FUNCTION_BLOCK FB_NTZ_KW
VAR_INPUT
	Freigabe_auto			: BOOL;
	Freigabe_Deakt_auto		: BOOL;
	Betrieb_Anford_auto		: BOOL;
	Regelung_Modus_auto		: SINT;
	Regelung_Sollw_auto		: REAL;
	Zustand_PSp				: ST_PSp_Zustand;
END_VAR
VAR_OUTPUT
END_VAR
VAR
	{attribute 'OPC.UA.DA' := '1'}Steuerung				: ST_ThNTZ_Steuerung;		
	{attribute 'OPC.UA.DA' := '1'}Stellwert				: ST_ThNTZ_Stellwert;		
	{attribute 'OPC.UA.DA' := '1'}Zustand					: ST_ThNTZ_Zustand;		
	{attribute 'OPC.UA.DA' := '1'}Parameter				: ST_ThNTZ_Parameter;		

	Zuweisungen             : FB_KW_Zuweisungen;
	Zustandscheck			: FB_ThNTZ_Zustandscheck;
	Logik					: FB_ThNTZ_Logik;
	Ablaufsteuerung			: FB_ThNTZ_Ablaufsteuerung;
	Sollwertscheck			: FB_ThNTZ_Sollwertscheck;
	Regelung				: FB_ThNTZ_Regelung_Kaltnetz;
	Stellwertscheck			: FB_ThNTZ_Stellwertscheck;
END_VAR

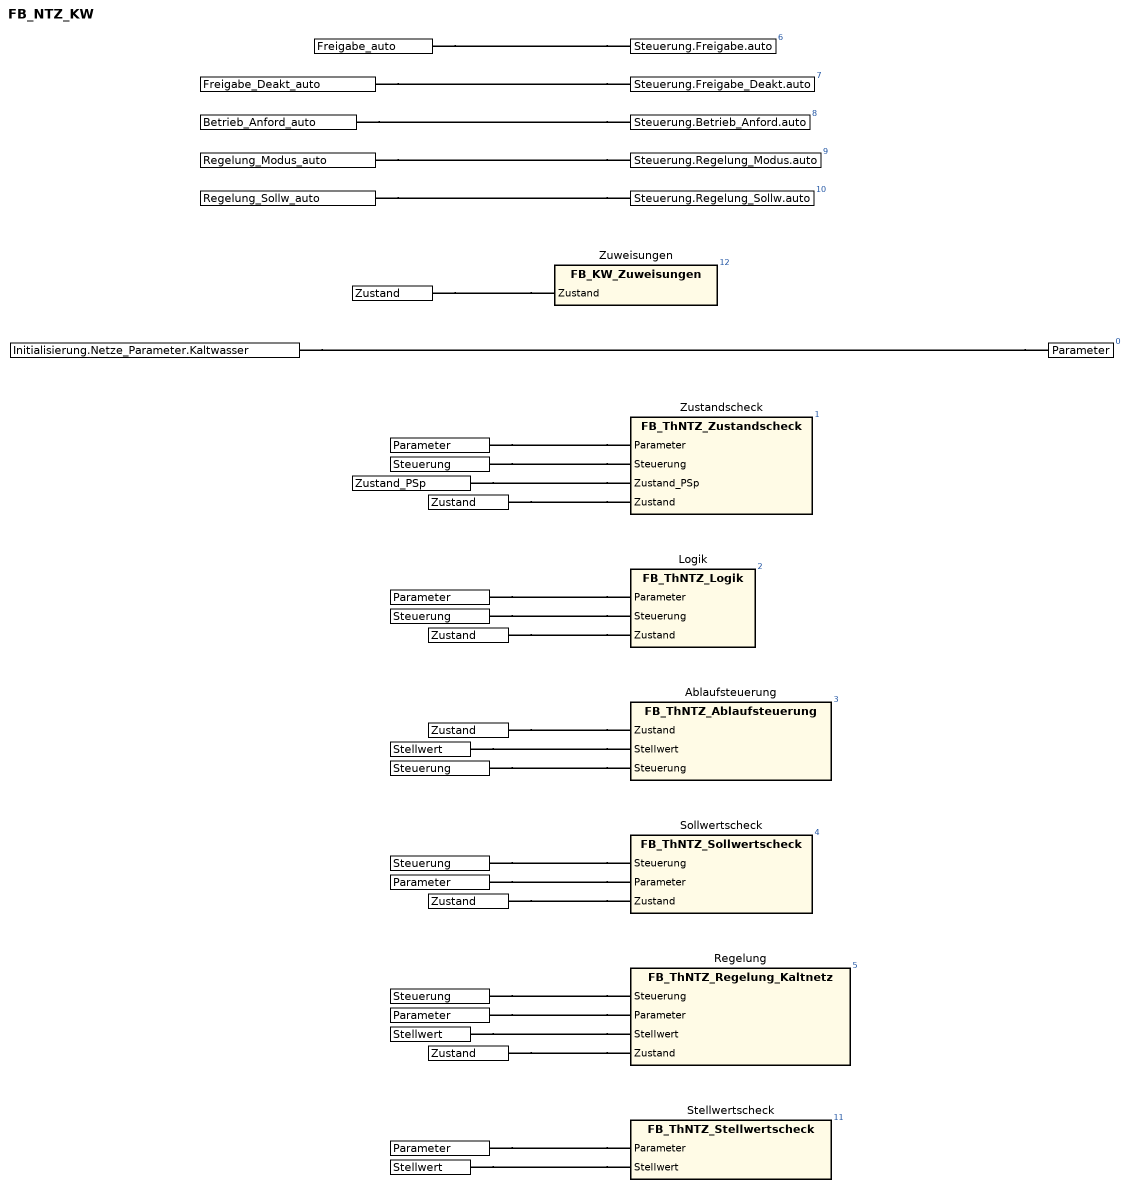
Parameter := Initialisierung.Netze_Parameter.Kaltwasser;
Zustandscheck(Parameter := Parameter, Steuerung := Steuerung, Zustand_PSp := Zustand_PSp, Zustand := Zustand); // FB_ThNTZ_Zustandscheck
Logik(Parameter := Parameter, Steuerung := Steuerung, Zustand := Zustand); // FB_ThNTZ_Logik
Ablaufsteuerung(Zustand := Zustand, Stellwert := Stellwert, Steuerung := Steuerung); // FB_ThNTZ_Ablaufsteuerung
Sollwertscheck(Steuerung := Steuerung, Parameter := Parameter, Zustand := Zustand); // FB_ThNTZ_Sollwertscheck
Regelung(Steuerung := Steuerung, Parameter := Parameter, Stellwert := Stellwert, Zustand := Zustand); // FB_ThNTZ_Regelung_Kaltnetz
Steuerung.Freigabe.auto := Freigabe_auto;
Steuerung.Freigabe_Deakt.auto := Freigabe_Deakt_auto;
Steuerung.Betrieb_Anford.auto := Betrieb_Anford_auto;
Steuerung.Regelung_Modus.auto := Regelung_Modus_auto;
Steuerung.Regelung_Sollw.auto := Regelung_Sollw_auto;
Stellwertscheck(Parameter := Parameter, Stellwert := Stellwert); // FB_ThNTZ_Stellwertscheck
Zuweisungen(Zustand := Zustand); // FB_KW_Zuweisungen

END_FUNCTION_BLOCK

(* stored: Version 1.1.0.1, ProductVersion 3.1.4024.9
   POU FB_NTZ_KW: Id {26cd2158-53ab-4dad-aa44-3e89f1ccca93}, SpecialFunc None *)
